// Mitsubishi GX Works2 project: plc_torque2   PLC: FX3U/FX3UC

PROGRAM MAIN
VAR
  __IST_dc39082d47ad4a44 : I+ST_dc39082d47ad4a44;
  __IST_c53a101abd94488d : I+ST_c53a101abd94488d;
END_VAR
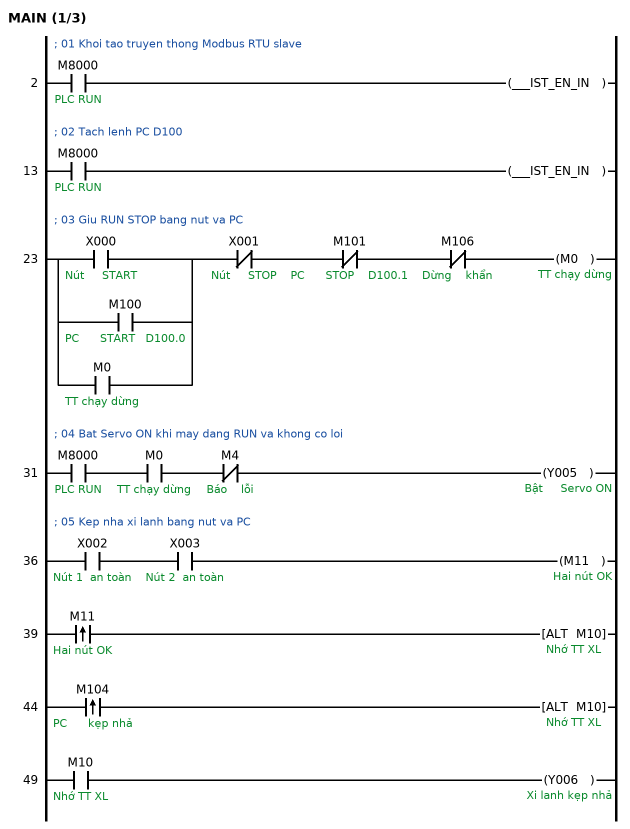
; FB BLK START I+ST_dc39082d47ad4a44(__IST_dc39082d47ad4a44)
; 01 Khoi tao truyen thong Modbus RTU slave
2     LD      M8000  ; PLC RUN
      OUT     ___IST_EN_IN
; FB START
; FB_NAME I+ST_dc39082d47ad4a44
; INSTANCE_NAME __IST_dc39082d47ad4a44
; FB IN_B:__IST_EN_IN
; FB OUT___IST_EN_OUT:B
; FB END
; FB BLK END
; 02 Tach lenh PC D100
; FB BLK START I+ST_c53a101abd94488d(__IST_c53a101abd94488d)
13    LD      M8000  ; PLC RUN
      OUT     ___IST_EN_IN
; FB START
; FB_NAME I+ST_c53a101abd94488d
; INSTANCE_NAME __IST_c53a101abd94488d
; FB IN_B:__IST_EN_IN
; FB OUT___IST_EN_OUT:B
; FB END
; FB BLK END
; 03 Giu RUN STOP bang nut va PC
23    LD      X000  ; Nút     START
      OR      M100  ; PC      START   D100.0
      OR      M0  ; TT chạy dừng
      ANI     X001  ; Nút     STOP
      ANI     M101  ; PC      STOP    D100.1
      ANI     M106  ; Dừng    khẩn
      OUT     M0  ; TT chạy dừng
; 04 Bat Servo ON khi may dang RUN va khong co loi
31    LD      M8000  ; PLC RUN
      AND     M0  ; TT chạy dừng
      ANI     M4  ; Báo    lỗi
      OUT     Y005  ; Bật     Servo ON
; 05 Kep nha xi lanh bang nut va PC
36    LD      X002  ; Nút 1  an toàn
      AND     X003  ; Nút 2  an toàn
      OUT     M11  ; Hai nút OK
39    LDP     M11  ; Hai nút OK
      ALT     M10  ; Nhớ TT XL
44    LDP     M104  ; PC      kẹp nhả
      ALT     M10
49    LD      M10  ; Nhớ TT XL
      OUT     Y006  ; Xi lanh kẹp nhả
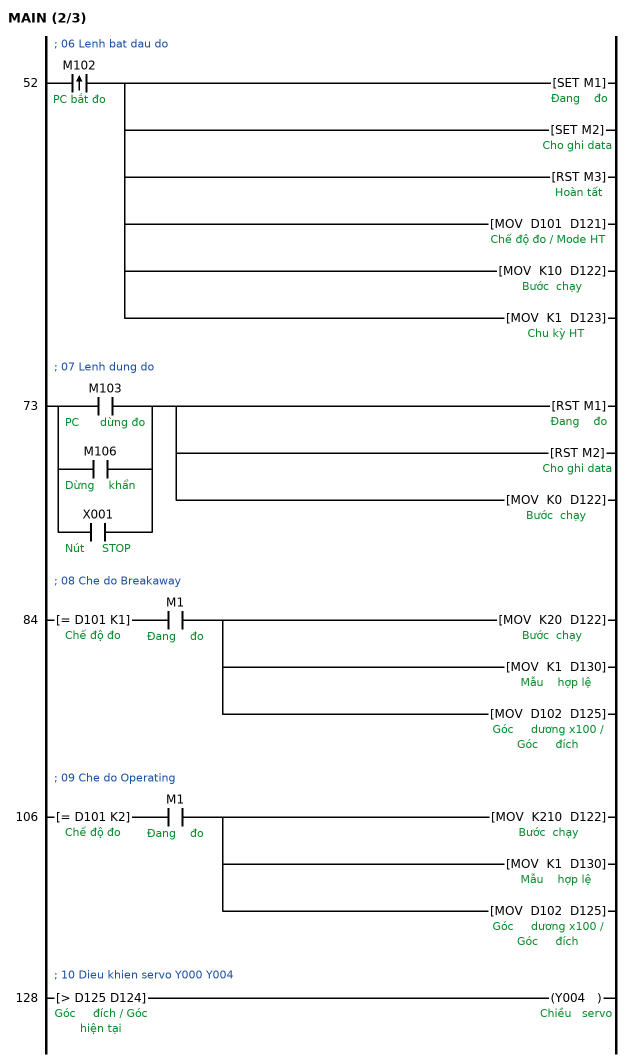
; 06 Lenh bat dau do
52    LDP     M102  ; PC bắt đo
      SET     M1  ; Đang    đo
      SET     M2  ; Cho ghi data
      RST     M3  ; Hoàn tất
      MOV     D101 D121  ; Chế độ đo / Mode HT
      MOV     K10 D122  ; Bước  chạy
      MOV     K1 D123  ; Chu kỳ HT
; 07 Lenh dung do
73    LD      M103  ; PC      dừng đo
      OR      M106  ; Dừng    khẩn
      OR      X001  ; Nút     STOP
      RST     M1  ; Đang    đo
      RST     M2  ; Cho ghi data
      MOV     K0 D122
; 08 Che do Breakaway
84    LD=     D101 K1  ; Chế độ đo
      AND     M1  ; Đang    đo
      MOV     K20 D122
      MOV     K1 D130  ; Mẫu    hợp lệ
      MOV     D102 D125  ; Góc     dương x100 / Góc     đích
; 09 Che do Operating
106   LD=     D101 K2  ; Chế độ đo
      AND     M1  ; Đang    đo
      MOV     K210 D122
      MOV     K1 D130
      MOV     D102 D125
; 10 Dieu khien servo Y000 Y004
128   LD>     D125 D124  ; Góc     đích / Góc     hiện tại
      OUT     Y004  ; Chiều   servo
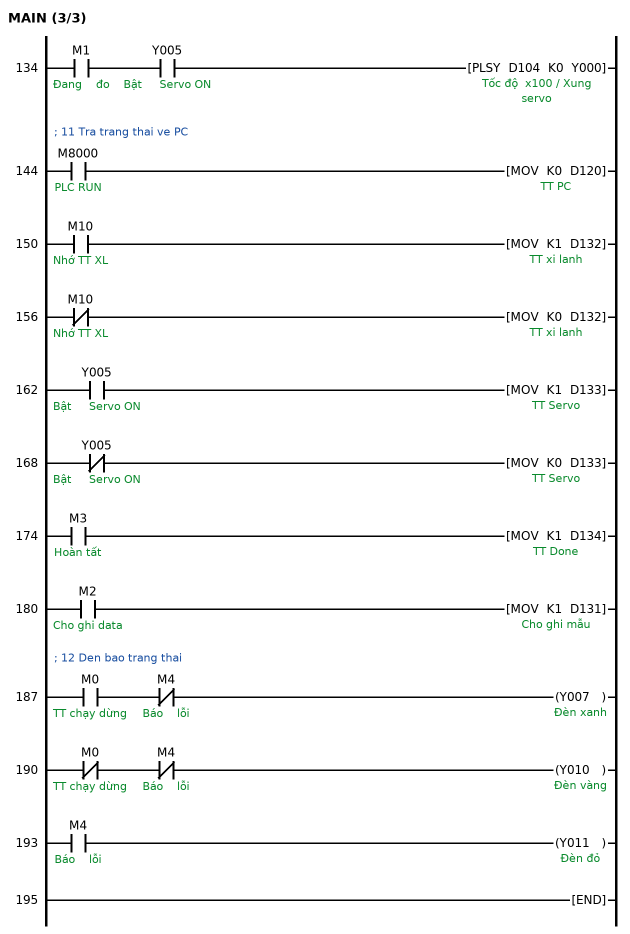
134   LD      M1  ; Đang    đo
      AND     Y005  ; Bật     Servo ON
      PLSY    D104 K0 Y000  ; Tốc độ  x100 / Xung    servo
; 11 Tra trang thai ve PC
144   LD      M8000  ; PLC RUN
      MOV     K0 D120  ; TT PC
150   LD      M10  ; Nhớ TT XL
      MOV     K1 D132  ; TT xi lanh
156   LDI     M10  ; Nhớ TT XL
      MOV     K0 D132
162   LD      Y005  ; Bật     Servo ON
      MOV     K1 D133  ; TT Servo
168   LDI     Y005  ; Bật     Servo ON
      MOV     K0 D133
174   LD      M3  ; Hoàn tất
      MOV     K1 D134  ; TT Done
180   LD      M2  ; Cho ghi data
      MOV     K1 D131  ; Cho ghi mẫu
; 12 Den bao trang thai
187   LD      M0  ; TT chạy dừng
      ANI     M4  ; Báo    lỗi
      OUT     Y007  ; Đèn xanh
190   LDI     M0  ; TT chạy dừng
      ANI     M4  ; Báo    lỗi
      OUT     Y010  ; Đèn vàng
193   LD      M4  ; Báo    lỗi
      OUT     Y011  ; Đèn đỏ
195   END
END_PROGRAM

FUNCTION_BLOCK I+ST_dc39082d47ad4a44
VAR_INPUT
  __IST_EN_IN : BOOL;
END_VAR
VAR_OUTPUT
  __IST_EN_OUT : BOOL;
END_VAR
(* IST HEADER START *)
IF NOT __IST_EN_IN THEN __IST_EN_OUT:=FALSE; RETURN; END_IF;
(* VERSION=1:TYPE=STB *)
(* IST HEADER END *)
(* FX3U Modbus RTU Slave - CH1 / 485ADP-MB *)

IF M8411 THEN
    D8400 := H10D1;   (* 8 bit, No parity, 1 stop, 115200 bps, RS485 *)
    D8401 := H0011;   (* Modbus Slave, RTU mode *)
    D8411 := K5;      (* message delay 5 ms *)
    D8414 := K2;      (* Slave ID = 2 *)
    D8415 := H0011;   (* lưu counter/log vào D *)
    D8416 := K100;    (* vùng status bắt đầu D100 *)
END_IF;
END_FUNCTION_BLOCK

FUNCTION_BLOCK I+ST_c53a101abd94488d
VAR_INPUT
  __IST_EN_IN : BOOL;
END_VAR
VAR_OUTPUT
  __IST_EN_OUT : BOOL;
END_VAR
(* IST HEADER START *)
IF NOT __IST_EN_IN THEN __IST_EN_OUT:=FALSE; RETURN; END_IF;
(* VERSION=1:TYPE=STB *)
(* IST HEADER END *)
M100 := D100.0;   (* PC START *)
M101 := D100.1;   (* PC STOP *)
M102 := D100.2;   (* PC bắt đầu *)
M103 := D100.3;   (* PC dừng đỏ *)
M104 := D100.4;   (* PC kẹp nhả *)
M105 := D100.5;   (* PC bật servo *)
M106 := D100.6;   (* Dừng khẩn *)
M107 := D100.7;   (* PC xóa DONE *)
END_FUNCTION_BLOCK

// device comments not shown above
M105  ; PC      bật servo
M107  ; PC      xóa    DONE
D100  ; Word    lệnh PC
D8400  ; 115200  8N1
D8401  ; Modbus  Slave   RTU
D8411  ; Delay   5 ms
D8414  ; Slave   ID bằng 2
D8415  ; Lưu D
D8416  ; Từ D100
M12  ; Xung 2 nút
M13  ; PC kẹp nhả
M20  ; Bắt ghi
M21  ; Dừng ghi
M30  ; SV đang chạy
M31  ; SV chạy xong
M32  ; SV chiều +
M33  ; SV chiều -
D103  ; Góc âm  x100
D105  ; Số chu kỳ
D106  ; Vùng    lấy mẫu
D107  ; Chọn    loại SP
D108  ; Loại    đo momen
D109  ; Reset   lỗi PC
D110  ; Jog     chiều dương
D111  ; Jog     chiều âm
D112  ; Lệnh    về gốc
D126  ; Tốc độ HT
D127  ; VT servo L
D128  ; VT servo H
D129  ; Mã lỗi  PLC
D135  ; Số mẫu
D150  ; Xung + L
D151  ; Xung + H
D152  ; Xung - L
D153  ; Xung - H
D154  ; Tốc xung L
D155  ; Tốc xung H
D156  ; Góc min OK
D157  ; Góc max OK
D158  ; TG bước
D160  ; Sai goc
D161  ; ABS goc
D162  ; Xung tinh L
D163  ; Xung tinh H
D164  ; So xung L
D165  ; So xung H
